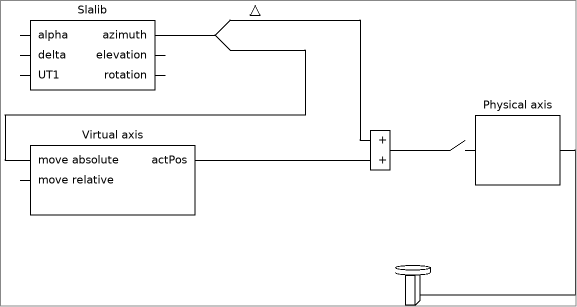
VISUALIZATION VISU_AxesRotationAxis_Overview  // 577x307
VAR_IN_OUT
	ref : AxesRotationAxis;
    widget : AxesRotationAxisWidget;
END_VAR
    Rectangle (405,275 10x30)
    Rectangle (30,20 125x70)
    Line (20,35) (30,35)
    Label (35,25 50x20), "alpha"
    Line (20,55) (30,55)
    Label (35,45 50x20), "delta"
    Line (20,75) (30,75)
    Label (35,65 50x20), "UT1"
    Polyline (255,5) (250,15) (260,15) (255,5)
    Label (30,0 125x20), "Slalib"
    Label (95,25 55x20), "azimuth"
    Label (90,45 60x20), "elevation"
    Label (100,65 50x20), "rotation"
    Line (155,55) (165,55)
    Line (155,75) (165,75)
    Rectangle (30,145 165x70)
    Label (35,150 95x20), "move absolute"
    Line (20,180) (30,180)
    Label (35,170 85x20), "move relative"
    Label (30,125 165x20), "Virtual axis"
    Label (135,150 55x20), "actPos"
    Polyline (155,35) (215,35) (230,50)
    Polyline (230,50) (305,50) (305,115) (5,115) (5,160) (30,160)
    Polyline (215,35) (230,20) (360,20) (360,140) (370,140)
    Polyline (195,160) (370,160)
    Rectangle (370,130 20x40)
    Label (375,130 15x20), "+"
    Label (375,150 15x20), "+"
    Line (390,150) (450,150)
    Line (450,150) (465,140)
    Line (465,150) (475,150)
    Rectangle (475,115 85x70)
    Label (475,95 85x20), "Physical axis"
    Polyline (560,150) (575,150) (575,295) (420,295)
    Polyline (415,305) (420,300) (420,275)
    Ellipse (395,270 35x5)
    Rectangle (395,270 35x2)
    Ellipse (395,265 35x5)
    Line (430,267) (430,272)
END_VISUALIZATION

(* stored: Version 1.1.0.1, ProductVersion 3.1.4019.2
   Visu VISU_AxesRotationAxis_Overview: Id {47a211cc-9b36-4ae8-9314-49e4f4b353e8} *)
